// TwinCAT 3 PLC project PLC
// ProgramVersion: 3.1.4026.26
// libraries:
//   Tc2_Standard, * (Beckhoff Automation GmbH)
//   Tc2_System, * (Beckhoff Automation GmbH)
// project tree:
//   GVLs/ IO_Main.TcGVL
//   / PlcTask.TcTTO
//   POUs/ MAIN.TcPOU
// real-time tasks:
//   TASK PlcTask: cycle T#10ms, priority 20, ADS port 350
// I/O:
//   DEVICE MAIN (EtherCAT), AmsNetId 192.168.0.103.2.1
//     Term 1 (EK1200) [EK1200-5000 EtherCAT Power supply (2A E-Bus)]
//       DI-01 (EL1809) [EL1809 16Ch. Dig. Input 24V, 3ms]
//       DI-02 (EL1809) [EL1809 16Ch. Dig. Input 24V, 3ms]
//       DO-01 (EL2809) [EL2809 16Ch. Dig. Output 24V, 0.5A]
//       DO-02 (EL2809) [EL2809 16Ch. Dig. Output 24V, 0.5A]
//       F-PLC (EL6910) [EL6910, TwinSAFE PLC]
//       FDI-01 (EL1918) [EL1918, 8Ch. Safety Input 24V, TwinSAFE]
//         modules: Module 1 (FSOE), Module 2 (FSLOGIC)
//       FDI-02 (EL1918) [EL1918, 8Ch. Safety Input 24V, TwinSAFE]
//         modules: Module 1 (FSOE), Module 2 (FSLOGIC)
//       FDO-01 (EL2912) [EL2912, 2Ch. Safety Output 24V, 2A, TwinSAFE]
//         modules: Module 1 (FSOE), Module 2 (FSOUT), Module 3 (DEVICEIO), Module 4 (FSLOGIC)
//       FDO-02 (EL2912) [EL2912, 2Ch. Safety Output 24V, 2A, TwinSAFE]
//         modules: Module 1 (FSOE), Module 2 (FSOUT), Module 3 (DEVICEIO), Module 4 (FSLOGIC)
//       POWER_SUPPLY (EL9410) [EL9410 E-Bus Power Supplier  (Diagnostics)]
//       PROFNET (EL6633) [EL6633 PROFINET IO Controller]
//       ETHERCAT (EK1322) [EK1322 2-port EtherCAT P junction with feed-in]
//       END_TERMINAL (EL9011) [EL9011 End Terminal]

CONFIGURATION PLC
    RESOURCE PLC ON TwinCAT3
        TASK PlcTask(INTERVAL := T#10ms, PRIORITY := 20);
        PROGRAM MAIN WITH PlcTask : MAIN;
    END_RESOURCE
END_CONFIGURATION

// ---- GVLs/IO_Main.TcGVL
{attribute 'qualified_only'}
VAR_GLOBAL
	//DI-01
	LM3_Fault AT%I*:BOOL;
	LM4_Fault AT%I*:BOOL;
	LM5_Fault AT%I*:BOOL;
	LM6_Fault AT%I*:BOOL;
	LM7_Fault AT%I*:BOOL;
	LM8_Fault AT%I*:BOOL;
	LM9_Fault AT%I*:BOOL;
	LM10_Fault AT%I*:BOOL;
	LM11_Fault AT%I*:BOOL;
	LM12_Fault AT%I*:BOOL;
	LM13_Fault AT%I*:BOOL;
	LM14_Fault AT%I*:BOOL;
	LM15_Fault AT%I*:BOOL;
	LM16_Fault AT%I*:BOOL;
	_3PS1_OUT_100 AT%I*:BOOL;
	_3PS1_DC_OK AT%I*:BOOL;
	
	//DI-02
	BACKUP_SIGNAL AT%I*:BOOL;
	TROUBLE_SIGNAL AT%I*:BOOL;
	BATTERY_LOW_SIGNAL AT%I*:BOOL;
	BATTERY_REPLACEMENT AT%I*:BOOL;
	
	//DO-01
	LM3_16_SET_RESET  AT%Q*:BOOL;
	_20K50_BEACON_INDICATOR_RED AT%Q*:BOOL;
	_20K50_BEACON_INDICATOR_YELLOW AT%Q*:BOOL;
	_20K50_BEACON_INDICATOR_GREEN AT%Q*:BOOL;
	_20K50_BEACON_INDICATOR_BUZZER AT%Q*:BOOL;
	
	//DO-02
	_3BPS1_REMOTE_ON_OFF AT%Q*:BOOL;
	_3BPS1_BACKUP_STOP AT%Q*:BOOL;
	
	//FDI-01
	EMERGENCY_STOP_ON_DOOR_CH1 AT%I*:BOOL;
	EMERGENCY_STOP_ON_DOOR_CH2 AT%I*:BOOL;
	RESET_ON_DOOR AT%I*:BOOL;
END_VAR

// ---- POUs/MAIN.TcPOU
PROGRAM MAIN
VAR
END_VAR

END_PROGRAM
